PROGRAM FertilizerProcess
VAR

(***********************************************Napedy w procesie produkcji nawozu z pofermentu i osadu****************************************************************************************)
	//Napedy U11 pompy SP02	
	fbDrvInv_SP02 		: FB_DriveInv(1, E_InvType.Schneider);
	fbDrvContrInv_SP02  : FB_DriveControl(fbDrvInv_SP02);

	//Napedy M01 M02 VR01 - schemat U71, U81	
	fbDrvInv_M01 		: FB_DriveInv(7, E_InvType.Schneider);
	fbDrvContrInv_M01   : FB_DriveControl(fbDrvInv_M01);
	
	fbDrvInv_M02 		: FB_DriveInv(8, E_InvType.Schneider);
	fbDrvContrInv_M02   : FB_DriveControl(fbDrvInv_M02);
	
	//Naped klapy M03 VR01 - schemat U91 
	fbDrvInv_M03 		: FB_DriveInv(9, E_InvType.Schneider);
	fbDrvContrInv_M03   : FB_DriveControl(fbDrvInv_M03);
	
	//Naped wentylator BL01
	fbDrv_BL01			: FB_Drive_1C();
	fbDrvContr_BL01		: FB_DriveControl(fbDrv_BL01);

	//Napedy podajnik SC-01 i SC02
	fbDrv_SC01			: FB_Drive_1C();
	fbDrvContr_SC01	    : FB_DriveControl(fbDrv_SC01);
	
	fbDrv_SC02			: FB_Drive_1C();
	fbDrvContr_SC02		: FB_DriveControl(fbDrv_SC02);
		
	//Napedy S01_E01 i S02_E02
	fbDrv_E01			: FB_Drive_1C();
	fbDrvContr_E01	    : FB_DriveControl(fbDrv_E01);
	
	fbDrv_E02			: FB_Drive_1C();
	fbDrvContr_E02		: FB_DriveControl(fbDrv_E02);
	


(***********************************************Czujniki w procesie produkcji nawozu z pofermentu i osadu****************************************************************************************)
	//Temp Sensor
	fbTempSens_H01	 	: FB_Scaling; //Czujnik temperatury w hali H01
	
	//Rotary Sensor
	fbRotarySens_S01	 : FB_DigitalSensNC; //Czujnik poziomu w silosien S01 typu NC
	fbRotarySens_S02	 : FB_DigitalSensNC; //Czujnik poziomu w silosien S02 typu NC



(*********************************************** Bloki Process Controlller****************************************************************************************)

	(************** Granulation controller **************************************************)
	fbGranulationProcess : FB_GranulationProcess;
	
	(************** Flap controller **************************************************)
	fbFlapControl		: FB_FlapCtrl; //controller bloku sterowania klapa
	

	
END_VAR
VAR // added by the converter: edge detectors and wires of the graphical bodies
    _w1, _w3, _w4 : ANY;
    _w2 : BOOL;
END_VAR

//Action
//Czujniki
ACT_WeightSensor(); //Sensor wagowy
ACT_TempSens();		//Sensor temperatury
ACT_DigitalSens();  //Sensory poziomu

//Automat nastawy napedów obsługi klapy
ACT_Control(); //Sterowanie procesem higienizacji

//Wybór nastawy napedów Auto lub SCADA
ACT_Motor(); //nastawy z SCADA



//**********************************SP-02*********************************************
//SP02
fbDrvContrInv_SP02();
GVL_Fertilizer.stDriveStatus_SP02 := fbDrvContrInv_SP02.StatusStruct(); //zwróc strukturę

//**********************************VR01*****************************************************
//M01
fbDrvContrInv_M01();
GVL_Fertilizer.stDriveStatus_M01 := fbDrvContrInv_M01.StatusStruct(); //zwróc strukturę
//M02
fbDrvContrInv_M02();
GVL_Fertilizer.stDriveStatus_M02 := fbDrvContrInv_M02.StatusStruct(); //zwróc strukturę
//M03
fbDrvContrInv_M03();
GVL_Fertilizer.stDriveStatus_M03 := fbDrvContrInv_M03.StatusStruct();

//**********************************Silosy S01 i S02*****************************************************
//SC01
fbDrvContr_SC01();
GVL_Fertilizer.stDriveStatus_SC01 := fbDrvContr_SC01.StatusStruct(); //zwróc strukturę
//SC02
fbDrvContr_SC02();
GVL_Fertilizer.stDriveStatus_SC02 := fbDrvContr_SC02.StatusStruct(); //zwróc strukturę
//E01
fbDrvContr_E01();
GVL_Fertilizer.stDriveStatus_E01 := fbDrvContr_E01.StatusStruct(); //zwróc strukturę
//E02
fbDrvContr_E02();
GVL_Fertilizer.stDriveStatus_E02 := fbDrvContr_E02.StatusStruct(); //zwróc strukturę

//**********************************BL01*****************************************************
//BL01
fbDrvContr_BL01();
GVL_Fertilizer.stDriveStatus_BL01 := fbDrvContr_BL01.StatusStruct(); //zwróc strukturę

ACTION ACT_Control:
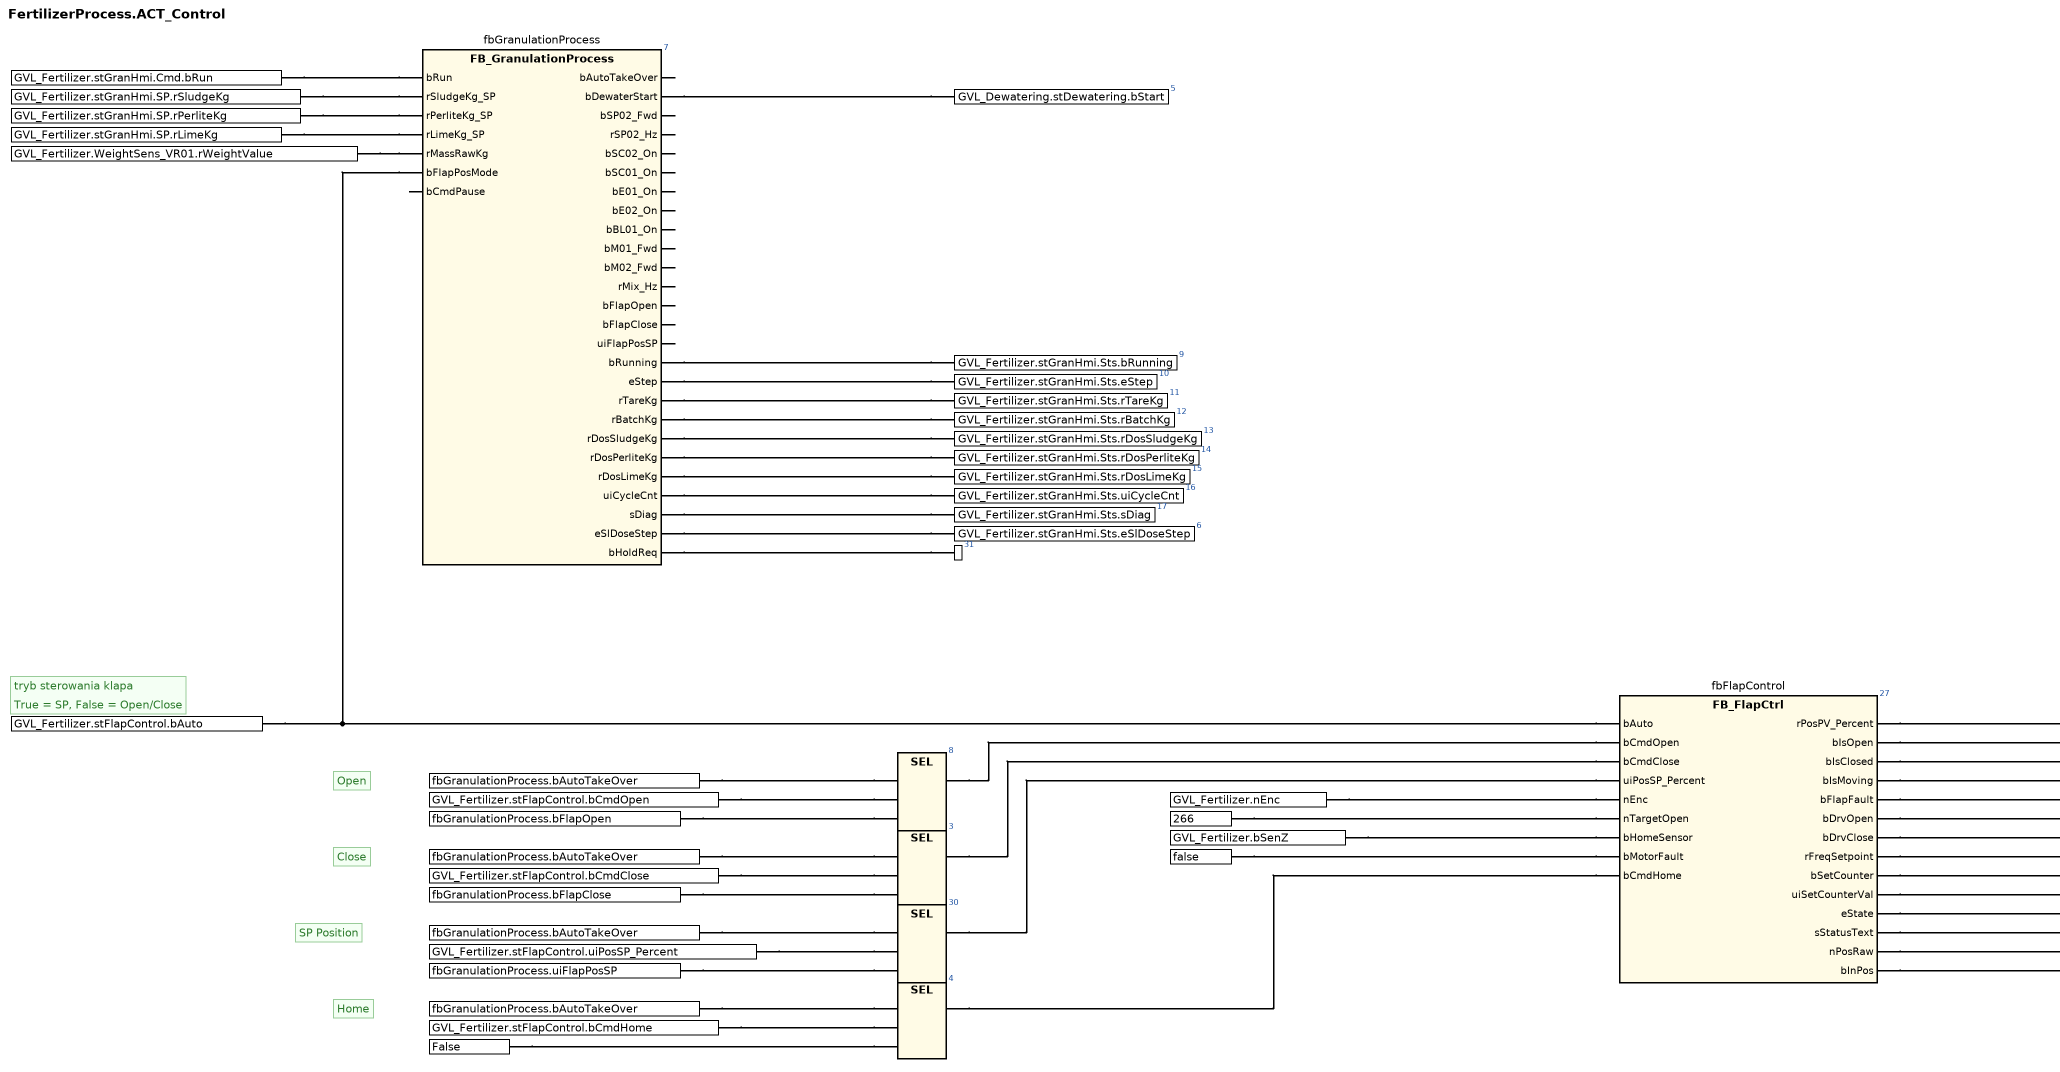
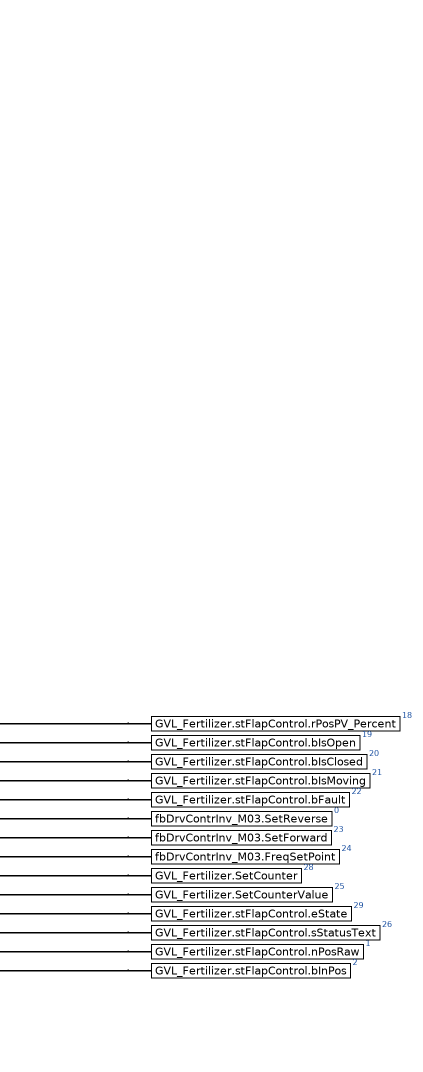
fbDrvContrInv_M03.SetReverse := fbFlapControl.bDrvOpen;
GVL_Fertilizer.stFlapControl.nPosRaw := fbFlapControl.nPosRaw;
GVL_Fertilizer.stFlapControl.bInPos := fbFlapControl.bInPos;
// Open
_w1 := SEL(fbGranulationProcess.bAutoTakeOver, GVL_Fertilizer.stFlapControl.bCmdClose, fbGranulationProcess.bFlapClose);
// SP Position
// Home
_w2 := SEL(fbGranulationProcess.bAutoTakeOver, GVL_Fertilizer.stFlapControl.bCmdHome, False);
GVL_Dewatering.stDewatering.bStart := fbGranulationProcess.bDewaterStart;
GVL_Fertilizer.stGranHmi.Sts.eSlDoseStep := fbGranulationProcess.eSlDoseStep;
fbGranulationProcess(
    bRun := GVL_Fertilizer.stGranHmi.Cmd.bRun,
    rSludgeKg_SP := GVL_Fertilizer.stGranHmi.SP.rSludgeKg,
    rPerliteKg_SP := GVL_Fertilizer.stGranHmi.SP.rPerliteKg,
    rLimeKg_SP := GVL_Fertilizer.stGranHmi.SP.rLimeKg,
    rMassRawKg := GVL_Fertilizer.WeightSens_VR01.rWeightValue,
    bFlapPosMode := GVL_Fertilizer.stFlapControl.bAuto); // FB_GranulationProcess
// tryb sterowania klapa
// True = SP, False = Open/Close
_w3 := SEL(fbGranulationProcess.bAutoTakeOver, GVL_Fertilizer.stFlapControl.bCmdOpen, fbGranulationProcess.bFlapOpen);
GVL_Fertilizer.stGranHmi.Sts.bRunning := fbGranulationProcess.bRunning;
GVL_Fertilizer.stGranHmi.Sts.eStep := fbGranulationProcess.eStep;
GVL_Fertilizer.stGranHmi.Sts.rTareKg := fbGranulationProcess.rTareKg;
GVL_Fertilizer.stGranHmi.Sts.rBatchKg := fbGranulationProcess.rBatchKg;
GVL_Fertilizer.stGranHmi.Sts.rDosSludgeKg := fbGranulationProcess.rDosSludgeKg;
GVL_Fertilizer.stGranHmi.Sts.rDosPerliteKg := fbGranulationProcess.rDosPerliteKg;
GVL_Fertilizer.stGranHmi.Sts.rDosLimeKg := fbGranulationProcess.rDosLimeKg;
GVL_Fertilizer.stGranHmi.Sts.uiCycleCnt := fbGranulationProcess.uiCycleCnt;
GVL_Fertilizer.stGranHmi.Sts.sDiag := fbGranulationProcess.sDiag;
GVL_Fertilizer.stFlapControl.rPosPV_Percent := fbFlapControl.rPosPV_Percent;
GVL_Fertilizer.stFlapControl.bIsOpen := fbFlapControl.bIsOpen;
GVL_Fertilizer.stFlapControl.bIsClosed := fbFlapControl.bIsClosed;
GVL_Fertilizer.stFlapControl.bIsMoving := fbFlapControl.bIsMoving;
GVL_Fertilizer.stFlapControl.bFault := fbFlapControl.bFlapFault;
fbDrvContrInv_M03.SetForward := fbFlapControl.bDrvClose;
fbDrvContrInv_M03.FreqSetPoint := fbFlapControl.rFreqSetpoint;
GVL_Fertilizer.SetCounterValue := fbFlapControl.uiSetCounterVal;
GVL_Fertilizer.stFlapControl.sStatusText := fbFlapControl.sStatusText;
fbFlapControl(
    bAuto := GVL_Fertilizer.stFlapControl.bAuto,
    bCmdOpen := _w3,
    bCmdClose := _w1,
    uiPosSP_Percent := _w4,
    nEnc := GVL_Fertilizer.nEnc,
    nTargetOpen := 266,
    bHomeSensor := GVL_Fertilizer.bSenZ,
    bMotorFault := false,
    bCmdHome := _w2); // FB_FlapCtrl
GVL_Fertilizer.SetCounter := fbFlapControl.bSetCounter;
GVL_Fertilizer.stFlapControl.eState := fbFlapControl.eState;
// Close
_w4 := SEL(fbGranulationProcess.bAutoTakeOver, GVL_Fertilizer.stFlapControl.uiPosSP_Percent, fbGranulationProcess.uiFlapPosSP);
??? := fbGranulationProcess.bHoldReq;
END_ACTION

ACTION ACT_DigitalSens:
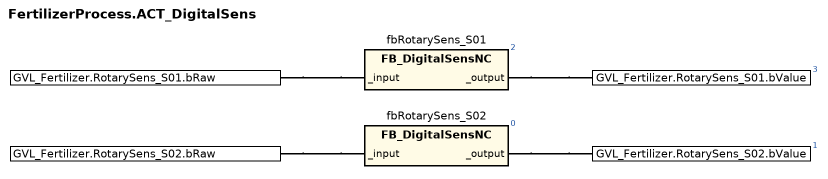
fbRotarySens_S02(_input := GVL_Fertilizer.RotarySens_S02.bRaw); // FB_DigitalSensNC
GVL_Fertilizer.RotarySens_S02.bValue := fbRotarySens_S02._output;
fbRotarySens_S01(_input := GVL_Fertilizer.RotarySens_S01.bRaw); // FB_DigitalSensNC
GVL_Fertilizer.RotarySens_S01.bValue := fbRotarySens_S01._output;
END_ACTION

ACTION ACT_Motor:

//************Naped ustawienia SP02**********************
//nastawy z SCADA lub z PLC blok nadrzędny wybór SELektorem
fbDrvContrInv_SP02.SetForward	:=SEL(fbGranulationProcess.bAutoTakeOver, GVL_Fertilizer.stDriveStatus_SP02.bForward, fbGranulationProcess.bSP02_Fwd);
fbDrvContrInv_SP02.SetReverse	:=SEL(fbGranulationProcess.bAutoTakeOver, GVL_Fertilizer.stDriveStatus_SP02.bReverse, FALSE); // w automacie nie ma reverse
fbDrvContrInv_SP02.FreqSetPoint	:=SEL(fbGranulationProcess.bAutoTakeOver, GVL_Fertilizer.stDriveStatus_SP02.FrequencySet, fbGranulationProcess.rSP02_Hz);

//***********Naped ustawienia VR01************************
//nastawy z SCADA M01 lub z PLC blok nadrzędny wybór SELektorem
fbDrvContrInv_M01.SetForward	:=SEL(fbGranulationProcess.bAutoTakeOver, GVL_Fertilizer.stDriveStatus_M01.bForward, fbGranulationProcess.bM01_Fwd);
fbDrvContrInv_M01.SetReverse	:=SEL(fbGranulationProcess.bAutoTakeOver, GVL_Fertilizer.stDriveStatus_M01.bReverse, FALSE);
fbDrvContrInv_M01.FreqSetPoint	:=SEL(fbGranulationProcess.bAutoTakeOver, GVL_Fertilizer.stDriveStatus_M01.FrequencySet, fbGranulationProcess.rMix_Hz);

//nastawy z SCADA M02 lub z PLC blok nadrzędny wybór SELektorem
fbDrvContrInv_M02.SetForward	:=SEL(fbGranulationProcess.bAutoTakeOver, GVL_Fertilizer.stDriveStatus_M02.bForward, fbGranulationProcess.bM02_Fwd);
fbDrvContrInv_M02.SetReverse	:=SEL(fbGranulationProcess.bAutoTakeOver, GVL_Fertilizer.stDriveStatus_M02.bReverse, FALSE);
fbDrvContrInv_M02.FreqSetPoint	:=SEL(fbGranulationProcess.bAutoTakeOver, GVL_Fertilizer.stDriveStatus_M02.FrequencySet, fbGranulationProcess.rMix_Hz);

//nastawy z SCADA M03
//fbDrvContrInv_M03.SetForward	:=GVL_Fertilizer.stDriveStatus_M03.bForward;
//fbDrvContrInv_M03.SetReverse	:=GVL_Fertilizer.stDriveStatus_M03.bReverse;
//fbDrvContrInv_M03.FreqSetPoint  :=GVL_Fertilizer.stDriveStatus_M03.FrequencySet;

//***********Naped ustawienia S01 i S02************************
//nastawy z SCADA SC01
fbDrvContr_SC01.SetForward	:=SEL(fbGranulationProcess.bAutoTakeOver, GVL_Fertilizer.stDriveStatus_SC01.bForward, fbGranulationProcess.bSC01_On);
//nastawy z SCADA SC02
fbDrvContr_SC02.SetForward	:=SEL(fbGranulationProcess.bAutoTakeOver, GVL_Fertilizer.stDriveStatus_SC02.bForward, fbGranulationProcess.bSC02_On);
//nastawy z SCADA E01
fbDrvContr_E01.SetForward	:=SEL(fbGranulationProcess.bAutoTakeOver, GVL_Fertilizer.stDriveStatus_E01.bForward, fbGranulationProcess.bE01_On);
//nastawy z SCADA E02
fbDrvContr_E02.SetForward	:=SEL(fbGranulationProcess.bAutoTakeOver, GVL_Fertilizer.stDriveStatus_E02.bForward, fbGranulationProcess.bE02_On);

////***********Naped ustawienia BL01 ************************
//nastawy z SCADA BL01
fbDrvContr_BL01.SetForward	:=SEL(fbGranulationProcess.bAutoTakeOver, GVL_Fertilizer.stDriveStatus_BL01.bForward, fbGranulationProcess.bBL01_On);
END_ACTION

ACTION ACT_TempSens:
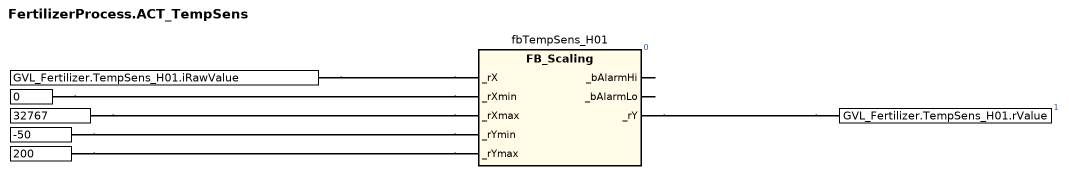
fbTempSens_H01(
    _rX := GVL_Fertilizer.TempSens_H01.iRawValue,
    _rXmin := 0,
    _rXmax := 32767,
    _rYmin := -50,
    _rYmax := 200); // FB_Scaling
GVL_Fertilizer.TempSens_H01.rValue := fbTempSens_H01._rY;
END_ACTION

ACTION ACT_WeightSensor:
//******************************************** Weight 01 ****************************************************
// WORD jest ze znakiem więc najpierw konwertujemy na INt aby otrzymac znak a potem na REAL

GVL_Fertilizer.WeightSens_VR01.rWeightValue := TO_REAL(TO_INT(GVL_Fertilizer.WeightSens_VR01.rRawWeightValue));
END_ACTION

END_PROGRAM

(* stored: Version 1.1.0.1, ProductVersion 3.1.4024.15
   POU FertilizerProcess: Id {ae9cea5e-de76-4d67-bab9-1dcc1d16bc80}, SpecialFunc None
   Action ACT_Control: Id {c00a6ec6-8960-40d8-ac4d-33202791525f}
   Action ACT_DigitalSens: Id {90fd9b42-e3eb-4636-915c-8178b327b54f}
   Action ACT_Motor: Id {157fa111-0c10-4c74-bf66-984a77c8c761}
   Action ACT_TempSens: Id {e5be406b-b6a0-4f64-8c1c-50c0deca9433}
   Action ACT_WeightSensor: Id {c3ec4534-bc74-4a01-b06c-42e2c4179453} *)
